{attribute 'linkalways'} 
{attribute 'no_explicit_call' := 'This FB is a CLASS and must be accessed using methods or properties'}
{attribute 'enable_dynamic_creation'}
FUNCTION_BLOCK PropertyAddedEvent EXTENDS Disposable IMPLEMENTS I_PropertyAddedEvent
VAR
	_targetProperty : I_Parameter;
END_VAR

METHOD FB_init : BOOL
VAR_INPUT
	bInitRetains : BOOL; // if TRUE, the retain variables are initialized (warm start / cold start)
	bInCopyCode : BOOL;  // if TRUE, the instance afterwards gets moved into the copy code (online change)
	TargetProperty : I_Parameter;
END_VAR
This^._targetProperty := TargetProperty;
END_METHOD

PROPERTY PUBLIC TargetProperty : I_Parameter
GET
TargetProperty := _targetProperty;
END_GET
END_PROPERTY

END_FUNCTION_BLOCK

(* stored: Version 1.1.0.1, ProductVersion 3.1.4024.12
   POU PropertyAddedEvent: Id {59b7d1eb-6f7f-02ba-2748-7daf463a196a}, SpecialFunc None
   Folder Constructor: Id {4e9e2852-6a90-07b7-223e-7b4ecb029181}
   Method FB_init: Id {6558aa10-c9cb-0c7c-0384-ea950b13cbaf}
   Property TargetProperty: Id {b3a818ea-dfe4-0faa-0ac2-b9bcdda27b4c}
   Get Get: Id {a636cc81-6e16-0bc5-3555-77caabe4b5f5} *)
